// Implicitly generated code : DO NOT EDIT
FUNCTION CheckLRangeUnsigned : ULINT
VAR_INPUT
	value, lower, upper: ULINT;
END_VAR

// Implicitly generated code: Only an implementation suggestion
IF (value < lower) THEN
	nCheckLRangeUnsigned := nCheckLRangeUnsigned + 1;
	CheckLRangeUnsigned := lower;
ELSIF(value > upper) THEN
	nCheckLRangeUnsigned := nCheckLRangeUnsigned + 1;
	CheckLRangeUnsigned := upper;
ELSE
	CheckLRangeUnsigned := value;
END_IF

END_FUNCTION

(* stored: Version 1.1.0.1
   POU CheckLRangeUnsigned: Id {8bed3751-07dd-4c7c-bad0-73a423200350}, SpecialFunc CheckLRangeUnsigned *)
